// TIA Portal V20 export
TYPE "LBP_typeTMTurret"
TITLE = Tool management / Gestion des outils
// User data type for block LBP_TMTurret [DB73] / Type de données utilisateur pour bloc LBP_TMTurret [DB73]
   STRUCT
      IFNo : Array[1..16] of Bool;   // Interface [number] active / Interface [numéro] active
      Quit : Array[1..16] of Bool;   // Perform Quit-End / Effectuer Quit-End
      TIF : Array[1..16] of Struct
         Comp : Bool;   // Compulsory change / Modification obligatoire
         Perform : Bool;   // Perform change / Effectuer modification/changement
         f0_2 : Bool;   // Reserved / Réservé
         T0 : Bool;   // T0 programmed / T0 programmé
         f0_4 : Bool;   // Reserved / Réservé
         f0_5 : Bool;   // Reserved / Réservé
         ManTOut : Bool;   // Unload hand tool from spindle manually / Décharger manuellement l'outil manuel de la broche
         f0_7 : Bool;   // Reserved / Réservé
         PerfStatusError : Bool;   // Negative acknowledge / Acquittement négatif
         n1_1 : Bool;   // Reserved / Réservé
         n1_2 : Bool;   // Reserved / Réservé
         n1_3 : Bool;   // Reserved / Réservé
         n1_4 : Bool;   // Reserved / Réservé
         n1_5 : Bool;   // Reserved / Réservé
         n1_6 : Bool;   // Reserved / Réservé
         DataInDB1073 : Bool;   // Multitool data stored in DB1073 / Données Multitool enregistrées dans DB1073
         Channel : Byte;   // Assigned channel / Canal affecté
         TMNo : Byte;   // Tool management number / Numéro de gestion des outils
         VdiTcp0 : DInt;   // User parameter 0 / Variable utilisateur libre 0
         VdiTcp1 : DInt;   // User parameter 1 / Variable utilisateur libre 1
         VdiTcp2 : DInt;   // User parameter 2 / Variable utilisateur libre 2
         BufferIdent : Int;   // Reserved (buffer identification) / Réservé (identifiant tampon)
         BufferNo : Int;   // Rel. location in buffer (res.) / Emplacement relatif dans tampon (rés.)
         SMag : Int;   // Magazine number of turret / Numéro de magasin de la tourelle
         SLoc : Int;   // Location number for new tool / Numéro d'emplacement du nouvel outil
         TMag : Int;   // Magazine number of turret (res.) / Numéro de magasin de la tourelle (rés.)
         TLoc : Int;   // Location number for previous tool / Numéro d'emplacement de l'outil précédent
         LocType : Int;   // Tool new: location type / Nouvel outil : type d'emplacement
         SLeft : Int;   // Tool new: size left / Nouvel outil : taille côté gauche
         SRight : Int;   // Tool new: size right / Nouvel outil : taille côté droit
         STop : Int;   // Tool new: size top / Nouvel outil : taille dessus
         SBottom : Int;   // Tool new: size bottom / Nouvel outil : taille dessous
         TInBuffer : Bool;   // ID for tools in buffer / ID pour outils dans tampon
         IgnoreDisabled : Bool;   // Ignore disabled / Ignorer désactivation
         Unload : Bool;   // To be unloaded / À décharger
         Load : Bool;   // To be loaded / À charger
         MasterTool : Bool;   // Tool is the master tool / L'outil est un outil principal
         n38_5 : Bool;   // Reserved / Réservé
         Exchange_1to1 : Bool;   // 1:1 exchange / Échange 1:1
         HandTool : Bool;   // Hand tool / Outil manuel
         Active : Bool;   // Active tool / Outil actif
         Enabled : Bool;   // Tool enabled / Outil activé
         Disabled : Bool;   // Tool disabled / Outil désactivé
         Measured : Bool;   // Tool measured / Outil mesuré
         Prewarn : Bool;   // Prewarning limit reached / Seuil de préavis atteint
         Change : Bool;   // Tool being changed / Outil en cours de changement
         FixedLoc : Bool;   // Tool fixed location coded / Emplacement fixe d'outil codé
         Used : Bool;   // Tool was in use / Outil a été utilisé
         TNo : Int;   // Tool new: T number / Nouvel outil : numéro d'outil
         MyPlace : Int;   // Original location of new tool / Emplacement d'origine du nouvel outil
      END_STRUCT;
   END_STRUCT;
   // // TIF[2].Comp : Compulsory change / Modification obligatoire
   // // TIF[3].Comp : Compulsory change / Modification obligatoire
   // // TIF[4].Comp : Compulsory change / Modification obligatoire
   // // TIF[5].Comp : Compulsory change / Modification obligatoire
   // // TIF[6].Comp : Compulsory change / Modification obligatoire
   // // TIF[7].Comp : Compulsory change / Modification obligatoire
   // // TIF[8].Comp : Compulsory change / Modification obligatoire
   // // TIF[9].Comp : Compulsory change / Modification obligatoire
   // // TIF[10].Comp : Compulsory change / Modification obligatoire
   // // TIF[11].Comp : Compulsory change / Modification obligatoire
   // // TIF[12].Comp : Compulsory change / Modification obligatoire
   // // TIF[13].Comp : Compulsory change / Modification obligatoire
   // // TIF[14].Comp : Compulsory change / Modification obligatoire
   // // TIF[15].Comp : Compulsory change / Modification obligatoire
   // // TIF[16].Comp : Compulsory change / Modification obligatoire
   // // TIF[2].Perform : Perform change / Effectuer modification/changement
   // // TIF[3].Perform : Perform change / Effectuer modification/changement
   // // TIF[4].Perform : Perform change / Effectuer modification/changement
   // // TIF[5].Perform : Perform change / Effectuer modification/changement
   // // TIF[6].Perform : Perform change / Effectuer modification/changement
   // // TIF[7].Perform : Perform change / Effectuer modification/changement
   // // TIF[8].Perform : Perform change / Effectuer modification/changement
   // // TIF[9].Perform : Perform change / Effectuer modification/changement
   // // TIF[10].Perform : Perform change / Effectuer modification/changement
   // // TIF[11].Perform : Perform change / Effectuer modification/changement
   // // TIF[12].Perform : Perform change / Effectuer modification/changement
   // // TIF[13].Perform : Perform change / Effectuer modification/changement
   // // TIF[14].Perform : Perform change / Effectuer modification/changement
   // // TIF[15].Perform : Perform change / Effectuer modification/changement
   // // TIF[16].Perform : Perform change / Effectuer modification/changement
   // // TIF[2].f0_2 : Reserved / Réservé
   // // TIF[3].f0_2 : Reserved / Réservé
   // // TIF[4].f0_2 : Reserved / Réservé
   // // TIF[5].f0_2 : Reserved / Réservé
   // // TIF[6].f0_2 : Reserved / Réservé
   // // TIF[7].f0_2 : Reserved / Réservé
   // // TIF[8].f0_2 : Reserved / Réservé
   // // TIF[9].f0_2 : Reserved / Réservé
   // // TIF[10].f0_2 : Reserved / Réservé
   // // TIF[11].f0_2 : Reserved / Réservé
   // // TIF[12].f0_2 : Reserved / Réservé
   // // TIF[13].f0_2 : Reserved / Réservé
   // // TIF[14].f0_2 : Reserved / Réservé
   // // TIF[15].f0_2 : Reserved / Réservé
   // // TIF[16].f0_2 : Reserved / Réservé
   // // TIF[2].T0 : T0 programmed / T0 programmé
   // // TIF[3].T0 : T0 programmed / T0 programmé
   // // TIF[4].T0 : T0 programmed / T0 programmé
   // // TIF[5].T0 : T0 programmed / T0 programmé
   // // TIF[6].T0 : T0 programmed / T0 programmé
   // // TIF[7].T0 : T0 programmed / T0 programmé
   // // TIF[8].T0 : T0 programmed / T0 programmé
   // // TIF[9].T0 : T0 programmed / T0 programmé
   // // TIF[10].T0 : T0 programmed / T0 programmé
   // // TIF[11].T0 : T0 programmed / T0 programmé
   // // TIF[12].T0 : T0 programmed / T0 programmé
   // // TIF[13].T0 : T0 programmed / T0 programmé
   // // TIF[14].T0 : T0 programmed / T0 programmé
   // // TIF[15].T0 : T0 programmed / T0 programmé
   // // TIF[16].T0 : T0 programmed / T0 programmé
   // // TIF[2].f0_4 : Reserved / Réservé
   // // TIF[3].f0_4 : Reserved / Réservé
   // // TIF[4].f0_4 : Reserved / Réservé
   // // TIF[5].f0_4 : Reserved / Réservé
   // // TIF[6].f0_4 : Reserved / Réservé
   // // TIF[7].f0_4 : Reserved / Réservé
   // // TIF[8].f0_4 : Reserved / Réservé
   // // TIF[9].f0_4 : Reserved / Réservé
   // // TIF[10].f0_4 : Reserved / Réservé
   // // TIF[11].f0_4 : Reserved / Réservé
   // // TIF[12].f0_4 : Reserved / Réservé
   // // TIF[13].f0_4 : Reserved / Réservé
   // // TIF[14].f0_4 : Reserved / Réservé
   // // TIF[15].f0_4 : Reserved / Réservé
   // // TIF[16].f0_4 : Reserved / Réservé
   // // TIF[2].f0_5 : Reserved / Réservé
   // // TIF[3].f0_5 : Reserved / Réservé
   // // TIF[4].f0_5 : Reserved / Réservé
   // // TIF[5].f0_5 : Reserved / Réservé
   // // TIF[6].f0_5 : Reserved / Réservé
   // // TIF[7].f0_5 : Reserved / Réservé
   // // TIF[8].f0_5 : Reserved / Réservé
   // // TIF[9].f0_5 : Reserved / Réservé
   // // TIF[10].f0_5 : Reserved / Réservé
   // // TIF[11].f0_5 : Reserved / Réservé
   // // TIF[12].f0_5 : Reserved / Réservé
   // // TIF[13].f0_5 : Reserved / Réservé
   // // TIF[14].f0_5 : Reserved / Réservé
   // // TIF[15].f0_5 : Reserved / Réservé
   // // TIF[16].f0_5 : Reserved / Réservé
   // // TIF[2].ManTOut : Unload hand tool from spindle manually / Décharger manuellement l'outil manuel de la broche
   // // TIF[3].ManTOut : Unload hand tool from spindle manually / Décharger manuellement l'outil manuel de la broche
   // // TIF[4].ManTOut : Unload hand tool from spindle manually / Décharger manuellement l'outil manuel de la broche
   // // TIF[5].ManTOut : Unload hand tool from spindle manually / Décharger manuellement l'outil manuel de la broche
   // // TIF[6].ManTOut : Unload hand tool from spindle manually / Décharger manuellement l'outil manuel de la broche
   // // TIF[7].ManTOut : Unload hand tool from spindle manually / Décharger manuellement l'outil manuel de la broche
   // // TIF[8].ManTOut : Unload hand tool from spindle manually / Décharger manuellement l'outil manuel de la broche
   // // TIF[9].ManTOut : Unload hand tool from spindle manually / Décharger manuellement l'outil manuel de la broche
   // // TIF[10].ManTOut : Unload hand tool from spindle manually / Décharger manuellement l'outil manuel de la broche
   // // TIF[11].ManTOut : Unload hand tool from spindle manually / Décharger manuellement l'outil manuel de la broche
   // // TIF[12].ManTOut : Unload hand tool from spindle manually / Décharger manuellement l'outil manuel de la broche
   // // TIF[13].ManTOut : Unload hand tool from spindle manually / Décharger manuellement l'outil manuel de la broche
   // // TIF[14].ManTOut : Unload hand tool from spindle manually / Décharger manuellement l'outil manuel de la broche
   // // TIF[15].ManTOut : Unload hand tool from spindle manually / Décharger manuellement l'outil manuel de la broche
   // // TIF[16].ManTOut : Unload hand tool from spindle manually / Décharger manuellement l'outil manuel de la broche
   // // TIF[2].f0_7 : Reserved / Réservé
   // // TIF[3].f0_7 : Reserved / Réservé
   // // TIF[4].f0_7 : Reserved / Réservé
   // // TIF[5].f0_7 : Reserved / Réservé
   // // TIF[6].f0_7 : Reserved / Réservé
   // // TIF[7].f0_7 : Reserved / Réservé
   // // TIF[8].f0_7 : Reserved / Réservé
   // // TIF[9].f0_7 : Reserved / Réservé
   // // TIF[10].f0_7 : Reserved / Réservé
   // // TIF[11].f0_7 : Reserved / Réservé
   // // TIF[12].f0_7 : Reserved / Réservé
   // // TIF[13].f0_7 : Reserved / Réservé
   // // TIF[14].f0_7 : Reserved / Réservé
   // // TIF[15].f0_7 : Reserved / Réservé
   // // TIF[16].f0_7 : Reserved / Réservé
   // // TIF[2].PerfStatusError : Negative acknowledge / Acquittement négatif
   // // TIF[3].PerfStatusError : Negative acknowledge / Acquittement négatif
   // // TIF[4].PerfStatusError : Negative acknowledge / Acquittement négatif
   // // TIF[5].PerfStatusError : Negative acknowledge / Acquittement négatif
   // // TIF[6].PerfStatusError : Negative acknowledge / Acquittement négatif
   // // TIF[7].PerfStatusError : Negative acknowledge / Acquittement négatif
   // // TIF[8].PerfStatusError : Negative acknowledge / Acquittement négatif
   // // TIF[9].PerfStatusError : Negative acknowledge / Acquittement négatif
   // // TIF[10].PerfStatusError : Negative acknowledge / Acquittement négatif
   // // TIF[11].PerfStatusError : Negative acknowledge / Acquittement négatif
   // // TIF[12].PerfStatusError : Negative acknowledge / Acquittement négatif
   // // TIF[13].PerfStatusError : Negative acknowledge / Acquittement négatif
   // // TIF[14].PerfStatusError : Negative acknowledge / Acquittement négatif
   // // TIF[15].PerfStatusError : Negative acknowledge / Acquittement négatif
   // // TIF[16].PerfStatusError : Negative acknowledge / Acquittement négatif
   // // TIF[2].n1_1 : Reserved / Réservé
   // // TIF[3].n1_1 : Reserved / Réservé
   // // TIF[4].n1_1 : Reserved / Réservé
   // // TIF[5].n1_1 : Reserved / Réservé
   // // TIF[6].n1_1 : Reserved / Réservé
   // // TIF[7].n1_1 : Reserved / Réservé
   // // TIF[8].n1_1 : Reserved / Réservé
   // // TIF[9].n1_1 : Reserved / Réservé
   // // TIF[10].n1_1 : Reserved / Réservé
   // // TIF[11].n1_1 : Reserved / Réservé
   // // TIF[12].n1_1 : Reserved / Réservé
   // // TIF[13].n1_1 : Reserved / Réservé
   // // TIF[14].n1_1 : Reserved / Réservé
   // // TIF[15].n1_1 : Reserved / Réservé
   // // TIF[16].n1_1 : Reserved / Réservé
   // // TIF[2].n1_2 : Reserved / Réservé
   // // TIF[3].n1_2 : Reserved / Réservé
   // // TIF[4].n1_2 : Reserved / Réservé
   // // TIF[5].n1_2 : Reserved / Réservé
   // // TIF[6].n1_2 : Reserved / Réservé
   // // TIF[7].n1_2 : Reserved / Réservé
   // // TIF[8].n1_2 : Reserved / Réservé
   // // TIF[9].n1_2 : Reserved / Réservé
   // // TIF[10].n1_2 : Reserved / Réservé
   // // TIF[11].n1_2 : Reserved / Réservé
   // // TIF[12].n1_2 : Reserved / Réservé
   // // TIF[13].n1_2 : Reserved / Réservé
   // // TIF[14].n1_2 : Reserved / Réservé
   // // TIF[15].n1_2 : Reserved / Réservé
   // // TIF[16].n1_2 : Reserved / Réservé
   // // TIF[2].n1_3 : Reserved / Réservé
   // // TIF[3].n1_3 : Reserved / Réservé
   // // TIF[4].n1_3 : Reserved / Réservé
   // // TIF[5].n1_3 : Reserved / Réservé
   // // TIF[6].n1_3 : Reserved / Réservé
   // // TIF[7].n1_3 : Reserved / Réservé
   // // TIF[8].n1_3 : Reserved / Réservé
   // // TIF[9].n1_3 : Reserved / Réservé
   // // TIF[10].n1_3 : Reserved / Réservé
   // // TIF[11].n1_3 : Reserved / Réservé
   // // TIF[12].n1_3 : Reserved / Réservé
   // // TIF[13].n1_3 : Reserved / Réservé
   // // TIF[14].n1_3 : Reserved / Réservé
   // // TIF[15].n1_3 : Reserved / Réservé
   // // TIF[16].n1_3 : Reserved / Réservé
   // // TIF[2].n1_4 : Reserved / Réservé
   // // TIF[3].n1_4 : Reserved / Réservé
   // // TIF[4].n1_4 : Reserved / Réservé
   // // TIF[5].n1_4 : Reserved / Réservé
   // // TIF[6].n1_4 : Reserved / Réservé
   // // TIF[7].n1_4 : Reserved / Réservé
   // // TIF[8].n1_4 : Reserved / Réservé
   // // TIF[9].n1_4 : Reserved / Réservé
   // // TIF[10].n1_4 : Reserved / Réservé
   // // TIF[11].n1_4 : Reserved / Réservé
   // // TIF[12].n1_4 : Reserved / Réservé
   // // TIF[13].n1_4 : Reserved / Réservé
   // // TIF[14].n1_4 : Reserved / Réservé
   // // TIF[15].n1_4 : Reserved / Réservé
   // // TIF[16].n1_4 : Reserved / Réservé
   // // TIF[2].n1_5 : Reserved / Réservé
   // // TIF[3].n1_5 : Reserved / Réservé
   // // TIF[4].n1_5 : Reserved / Réservé
   // // TIF[5].n1_5 : Reserved / Réservé
   // // TIF[6].n1_5 : Reserved / Réservé
   // // TIF[7].n1_5 : Reserved / Réservé
   // // TIF[8].n1_5 : Reserved / Réservé
   // // TIF[9].n1_5 : Reserved / Réservé
   // // TIF[10].n1_5 : Reserved / Réservé
   // // TIF[11].n1_5 : Reserved / Réservé
   // // TIF[12].n1_5 : Reserved / Réservé
   // // TIF[13].n1_5 : Reserved / Réservé
   // // TIF[14].n1_5 : Reserved / Réservé
   // // TIF[15].n1_5 : Reserved / Réservé
   // // TIF[16].n1_5 : Reserved / Réservé
   // // TIF[2].n1_6 : Reserved / Réservé
   // // TIF[3].n1_6 : Reserved / Réservé
   // // TIF[4].n1_6 : Reserved / Réservé
   // // TIF[5].n1_6 : Reserved / Réservé
   // // TIF[6].n1_6 : Reserved / Réservé
   // // TIF[7].n1_6 : Reserved / Réservé
   // // TIF[8].n1_6 : Reserved / Réservé
   // // TIF[9].n1_6 : Reserved / Réservé
   // // TIF[10].n1_6 : Reserved / Réservé
   // // TIF[11].n1_6 : Reserved / Réservé
   // // TIF[12].n1_6 : Reserved / Réservé
   // // TIF[13].n1_6 : Reserved / Réservé
   // // TIF[14].n1_6 : Reserved / Réservé
   // // TIF[15].n1_6 : Reserved / Réservé
   // // TIF[16].n1_6 : Reserved / Réservé
   // // TIF[2].DataInDB1073 : Multitool data stored in DB1073 / Données Multitool enregistrées dans DB1073
   // // TIF[3].DataInDB1073 : Multitool data stored in DB1073 / Données Multitool enregistrées dans DB1073
   // // TIF[4].DataInDB1073 : Multitool data stored in DB1073 / Données Multitool enregistrées dans DB1073
   // // TIF[5].DataInDB1073 : Multitool data stored in DB1073 / Données Multitool enregistrées dans DB1073
   // // TIF[6].DataInDB1073 : Multitool data stored in DB1073 / Données Multitool enregistrées dans DB1073
   // // TIF[7].DataInDB1073 : Multitool data stored in DB1073 / Données Multitool enregistrées dans DB1073
   // // TIF[8].DataInDB1073 : Multitool data stored in DB1073 / Données Multitool enregistrées dans DB1073
   // // TIF[9].DataInDB1073 : Multitool data stored in DB1073 / Données Multitool enregistrées dans DB1073
   // // TIF[10].DataInDB1073 : Multitool data stored in DB1073 / Données Multitool enregistrées dans DB1073
   // // TIF[11].DataInDB1073 : Multitool data stored in DB1073 / Données Multitool enregistrées dans DB1073
   // // TIF[12].DataInDB1073 : Multitool data stored in DB1073 / Données Multitool enregistrées dans DB1073
   // // TIF[13].DataInDB1073 : Multitool data stored in DB1073 / Données Multitool enregistrées dans DB1073
   // // TIF[14].DataInDB1073 : Multitool data stored in DB1073 / Données Multitool enregistrées dans DB1073
   // // TIF[15].DataInDB1073 : Multitool data stored in DB1073 / Données Multitool enregistrées dans DB1073
   // // TIF[16].DataInDB1073 : Multitool data stored in DB1073 / Données Multitool enregistrées dans DB1073
   // // TIF[2].Channel : Assigned channel / Canal affecté
   // // TIF[3].Channel : Assigned channel / Canal affecté
   // // TIF[4].Channel : Assigned channel / Canal affecté
   // // TIF[5].Channel : Assigned channel / Canal affecté
   // // TIF[6].Channel : Assigned channel / Canal affecté
   // // TIF[7].Channel : Assigned channel / Canal affecté
   // // TIF[8].Channel : Assigned channel / Canal affecté
   // // TIF[9].Channel : Assigned channel / Canal affecté
   // // TIF[10].Channel : Assigned channel / Canal affecté
   // // TIF[11].Channel : Assigned channel / Canal affecté
   // // TIF[12].Channel : Assigned channel / Canal affecté
   // // TIF[13].Channel : Assigned channel / Canal affecté
   // // TIF[14].Channel : Assigned channel / Canal affecté
   // // TIF[15].Channel : Assigned channel / Canal affecté
   // // TIF[16].Channel : Assigned channel / Canal affecté
   // // TIF[2].TMNo : Tool management number / Numéro de gestion des outils
   // // TIF[3].TMNo : Tool management number / Numéro de gestion des outils
   // // TIF[4].TMNo : Tool management number / Numéro de gestion des outils
   // // TIF[5].TMNo : Tool management number / Numéro de gestion des outils
   // // TIF[6].TMNo : Tool management number / Numéro de gestion des outils
   // // TIF[7].TMNo : Tool management number / Numéro de gestion des outils
   // // TIF[8].TMNo : Tool management number / Numéro de gestion des outils
   // // TIF[9].TMNo : Tool management number / Numéro de gestion des outils
   // // TIF[10].TMNo : Tool management number / Numéro de gestion des outils
   // // TIF[11].TMNo : Tool management number / Numéro de gestion des outils
   // // TIF[12].TMNo : Tool management number / Numéro de gestion des outils
   // // TIF[13].TMNo : Tool management number / Numéro de gestion des outils
   // // TIF[14].TMNo : Tool management number / Numéro de gestion des outils
   // // TIF[15].TMNo : Tool management number / Numéro de gestion des outils
   // // TIF[16].TMNo : Tool management number / Numéro de gestion des outils
   // // TIF[2].VdiTcp0 : User parameter 0 / Variable utilisateur libre 0
   // // TIF[3].VdiTcp0 : User parameter 0 / Variable utilisateur libre 0
   // // TIF[4].VdiTcp0 : User parameter 0 / Variable utilisateur libre 0
   // // TIF[5].VdiTcp0 : User parameter 0 / Variable utilisateur libre 0
   // // TIF[6].VdiTcp0 : User parameter 0 / Variable utilisateur libre 0
   // // TIF[7].VdiTcp0 : User parameter 0 / Variable utilisateur libre 0
   // // TIF[8].VdiTcp0 : User parameter 0 / Variable utilisateur libre 0
   // // TIF[9].VdiTcp0 : User parameter 0 / Variable utilisateur libre 0
   // // TIF[10].VdiTcp0 : User parameter 0 / Variable utilisateur libre 0
   // // TIF[11].VdiTcp0 : User parameter 0 / Variable utilisateur libre 0
   // // TIF[12].VdiTcp0 : User parameter 0 / Variable utilisateur libre 0
   // // TIF[13].VdiTcp0 : User parameter 0 / Variable utilisateur libre 0
   // // TIF[14].VdiTcp0 : User parameter 0 / Variable utilisateur libre 0
   // // TIF[15].VdiTcp0 : User parameter 0 / Variable utilisateur libre 0
   // // TIF[16].VdiTcp0 : User parameter 0 / Variable utilisateur libre 0
   // // TIF[2].VdiTcp1 : User parameter 1 / Variable utilisateur libre 1
   // // TIF[3].VdiTcp1 : User parameter 1 / Variable utilisateur libre 1
   // // TIF[4].VdiTcp1 : User parameter 1 / Variable utilisateur libre 1
   // // TIF[5].VdiTcp1 : User parameter 1 / Variable utilisateur libre 1
   // // TIF[6].VdiTcp1 : User parameter 1 / Variable utilisateur libre 1
   // // TIF[7].VdiTcp1 : User parameter 1 / Variable utilisateur libre 1
   // // TIF[8].VdiTcp1 : User parameter 1 / Variable utilisateur libre 1
   // // TIF[9].VdiTcp1 : User parameter 1 / Variable utilisateur libre 1
   // // TIF[10].VdiTcp1 : User parameter 1 / Variable utilisateur libre 1
   // // TIF[11].VdiTcp1 : User parameter 1 / Variable utilisateur libre 1
   // // TIF[12].VdiTcp1 : User parameter 1 / Variable utilisateur libre 1
   // // TIF[13].VdiTcp1 : User parameter 1 / Variable utilisateur libre 1
   // // TIF[14].VdiTcp1 : User parameter 1 / Variable utilisateur libre 1
   // // TIF[15].VdiTcp1 : User parameter 1 / Variable utilisateur libre 1
   // // TIF[16].VdiTcp1 : User parameter 1 / Variable utilisateur libre 1
   // // TIF[2].VdiTcp2 : User parameter 2 / Variable utilisateur libre 2
   // // TIF[3].VdiTcp2 : User parameter 2 / Variable utilisateur libre 2
   // // TIF[4].VdiTcp2 : User parameter 2 / Variable utilisateur libre 2
   // // TIF[5].VdiTcp2 : User parameter 2 / Variable utilisateur libre 2
   // // TIF[6].VdiTcp2 : User parameter 2 / Variable utilisateur libre 2
   // // TIF[7].VdiTcp2 : User parameter 2 / Variable utilisateur libre 2
   // // TIF[8].VdiTcp2 : User parameter 2 / Variable utilisateur libre 2
   // // TIF[9].VdiTcp2 : User parameter 2 / Variable utilisateur libre 2
   // // TIF[10].VdiTcp2 : User parameter 2 / Variable utilisateur libre 2
   // // TIF[11].VdiTcp2 : User parameter 2 / Variable utilisateur libre 2
   // // TIF[12].VdiTcp2 : User parameter 2 / Variable utilisateur libre 2
   // // TIF[13].VdiTcp2 : User parameter 2 / Variable utilisateur libre 2
   // // TIF[14].VdiTcp2 : User parameter 2 / Variable utilisateur libre 2
   // // TIF[15].VdiTcp2 : User parameter 2 / Variable utilisateur libre 2
   // // TIF[16].VdiTcp2 : User parameter 2 / Variable utilisateur libre 2
   // // TIF[2].BufferIdent : Reserved (buffer identification) / Réservé (identifiant tampon)
   // // TIF[3].BufferIdent : Reserved (buffer identification) / Réservé (identifiant tampon)
   // // TIF[4].BufferIdent : Reserved (buffer identification) / Réservé (identifiant tampon)
   // // TIF[5].BufferIdent : Reserved (buffer identification) / Réservé (identifiant tampon)
   // // TIF[6].BufferIdent : Reserved (buffer identification) / Réservé (identifiant tampon)
   // // TIF[7].BufferIdent : Reserved (buffer identification) / Réservé (identifiant tampon)
   // // TIF[8].BufferIdent : Reserved (buffer identification) / Réservé (identifiant tampon)
   // // TIF[9].BufferIdent : Reserved (buffer identification) / Réservé (identifiant tampon)
   // // TIF[10].BufferIdent : Reserved (buffer identification) / Réservé (identifiant tampon)
   // // TIF[11].BufferIdent : Reserved (buffer identification) / Réservé (identifiant tampon)
   // // TIF[12].BufferIdent : Reserved (buffer identification) / Réservé (identifiant tampon)
   // // TIF[13].BufferIdent : Reserved (buffer identification) / Réservé (identifiant tampon)
   // // TIF[14].BufferIdent : Reserved (buffer identification) / Réservé (identifiant tampon)
   // // TIF[15].BufferIdent : Reserved (buffer identification) / Réservé (identifiant tampon)
   // // TIF[16].BufferIdent : Reserved (buffer identification) / Réservé (identifiant tampon)
   // // TIF[2].BufferNo : Rel. location in buffer (res.) / Emplacement relatif dans tampon (rés.)
   // // TIF[3].BufferNo : Rel. location in buffer (res.) / Emplacement relatif dans tampon (rés.)
   // // TIF[4].BufferNo : Rel. location in buffer (res.) / Emplacement relatif dans tampon (rés.)
   // // TIF[5].BufferNo : Rel. location in buffer (res.) / Emplacement relatif dans tampon (rés.)
   // // TIF[6].BufferNo : Rel. location in buffer (res.) / Emplacement relatif dans tampon (rés.)
   // // TIF[7].BufferNo : Rel. location in buffer (res.) / Emplacement relatif dans tampon (rés.)
   // // TIF[8].BufferNo : Rel. location in buffer (res.) / Emplacement relatif dans tampon (rés.)
   // // TIF[9].BufferNo : Rel. location in buffer (res.) / Emplacement relatif dans tampon (rés.)
   // // TIF[10].BufferNo : Rel. location in buffer (res.) / Emplacement relatif dans tampon (rés.)
   // // TIF[11].BufferNo : Rel. location in buffer (res.) / Emplacement relatif dans tampon (rés.)
   // // TIF[12].BufferNo : Rel. location in buffer (res.) / Emplacement relatif dans tampon (rés.)
   // // TIF[13].BufferNo : Rel. location in buffer (res.) / Emplacement relatif dans tampon (rés.)
   // // TIF[14].BufferNo : Rel. location in buffer (res.) / Emplacement relatif dans tampon (rés.)
   // // TIF[15].BufferNo : Rel. location in buffer (res.) / Emplacement relatif dans tampon (rés.)
   // // TIF[16].BufferNo : Rel. location in buffer (res.) / Emplacement relatif dans tampon (rés.)
   // // TIF[2].SMag : Magazine number of turret / Numéro de magasin de la tourelle
   // // TIF[3].SMag : Magazine number of turret / Numéro de magasin de la tourelle
   // // TIF[4].SMag : Magazine number of turret / Numéro de magasin de la tourelle
   // // TIF[5].SMag : Magazine number of turret / Numéro de magasin de la tourelle
   // // TIF[6].SMag : Magazine number of turret / Numéro de magasin de la tourelle
   // // TIF[7].SMag : Magazine number of turret / Numéro de magasin de la tourelle
   // // TIF[8].SMag : Magazine number of turret / Numéro de magasin de la tourelle
   // // TIF[9].SMag : Magazine number of turret / Numéro de magasin de la tourelle
   // // TIF[10].SMag : Magazine number of turret / Numéro de magasin de la tourelle
   // // TIF[11].SMag : Magazine number of turret / Numéro de magasin de la tourelle
   // // TIF[12].SMag : Magazine number of turret / Numéro de magasin de la tourelle
   // // TIF[13].SMag : Magazine number of turret / Numéro de magasin de la tourelle
   // // TIF[14].SMag : Magazine number of turret / Numéro de magasin de la tourelle
   // // TIF[15].SMag : Magazine number of turret / Numéro de magasin de la tourelle
   // // TIF[16].SMag : Magazine number of turret / Numéro de magasin de la tourelle
   // // TIF[2].SLoc : Location number for new tool / Numéro d'emplacement du nouvel outil
   // // TIF[3].SLoc : Location number for new tool / Numéro d'emplacement du nouvel outil
   // // TIF[4].SLoc : Location number for new tool / Numéro d'emplacement du nouvel outil
   // // TIF[5].SLoc : Location number for new tool / Numéro d'emplacement du nouvel outil
   // // TIF[6].SLoc : Location number for new tool / Numéro d'emplacement du nouvel outil
   // // TIF[7].SLoc : Location number for new tool / Numéro d'emplacement du nouvel outil
   // // TIF[8].SLoc : Location number for new tool / Numéro d'emplacement du nouvel outil
   // // TIF[9].SLoc : Location number for new tool / Numéro d'emplacement du nouvel outil
   // // TIF[10].SLoc : Location number for new tool / Numéro d'emplacement du nouvel outil
   // // TIF[11].SLoc : Location number for new tool / Numéro d'emplacement du nouvel outil
   // // TIF[12].SLoc : Location number for new tool / Numéro d'emplacement du nouvel outil
   // // TIF[13].SLoc : Location number for new tool / Numéro d'emplacement du nouvel outil
   // // TIF[14].SLoc : Location number for new tool / Numéro d'emplacement du nouvel outil
   // // TIF[15].SLoc : Location number for new tool / Numéro d'emplacement du nouvel outil
   // // TIF[16].SLoc : Location number for new tool / Numéro d'emplacement du nouvel outil
   // // TIF[2].TMag : Magazine number of turret (res.) / Numéro de magasin de la tourelle (rés.)
   // // TIF[3].TMag : Magazine number of turret (res.) / Numéro de magasin de la tourelle (rés.)
   // // TIF[4].TMag : Magazine number of turret (res.) / Numéro de magasin de la tourelle (rés.)
   // // TIF[5].TMag : Magazine number of turret (res.) / Numéro de magasin de la tourelle (rés.)
   // // TIF[6].TMag : Magazine number of turret (res.) / Numéro de magasin de la tourelle (rés.)
   // // TIF[7].TMag : Magazine number of turret (res.) / Numéro de magasin de la tourelle (rés.)
   // // TIF[8].TMag : Magazine number of turret (res.) / Numéro de magasin de la tourelle (rés.)
   // // TIF[9].TMag : Magazine number of turret (res.) / Numéro de magasin de la tourelle (rés.)
   // // TIF[10].TMag : Magazine number of turret (res.) / Numéro de magasin de la tourelle (rés.)
   // // TIF[11].TMag : Magazine number of turret (res.) / Numéro de magasin de la tourelle (rés.)
   // // TIF[12].TMag : Magazine number of turret (res.) / Numéro de magasin de la tourelle (rés.)
   // // TIF[13].TMag : Magazine number of turret (res.) / Numéro de magasin de la tourelle (rés.)
   // // TIF[14].TMag : Magazine number of turret (res.) / Numéro de magasin de la tourelle (rés.)
   // // TIF[15].TMag : Magazine number of turret (res.) / Numéro de magasin de la tourelle (rés.)
   // // TIF[16].TMag : Magazine number of turret (res.) / Numéro de magasin de la tourelle (rés.)
   // // TIF[2].TLoc : Location number for previous tool / Numéro d'emplacement de l'outil précédent
   // // TIF[3].TLoc : Location number for previous tool / Numéro d'emplacement de l'outil précédent
   // // TIF[4].TLoc : Location number for previous tool / Numéro d'emplacement de l'outil précédent
   // // TIF[5].TLoc : Location number for previous tool / Numéro d'emplacement de l'outil précédent
   // // TIF[6].TLoc : Location number for previous tool / Numéro d'emplacement de l'outil précédent
   // // TIF[7].TLoc : Location number for previous tool / Numéro d'emplacement de l'outil précédent
   // // TIF[8].TLoc : Location number for previous tool / Numéro d'emplacement de l'outil précédent
   // // TIF[9].TLoc : Location number for previous tool / Numéro d'emplacement de l'outil précédent
   // // TIF[10].TLoc : Location number for previous tool / Numéro d'emplacement de l'outil précédent
   // // TIF[11].TLoc : Location number for previous tool / Numéro d'emplacement de l'outil précédent
   // // TIF[12].TLoc : Location number for previous tool / Numéro d'emplacement de l'outil précédent
   // // TIF[13].TLoc : Location number for previous tool / Numéro d'emplacement de l'outil précédent
   // // TIF[14].TLoc : Location number for previous tool / Numéro d'emplacement de l'outil précédent
   // // TIF[15].TLoc : Location number for previous tool / Numéro d'emplacement de l'outil précédent
   // // TIF[16].TLoc : Location number for previous tool / Numéro d'emplacement de l'outil précédent
   // // TIF[2].LocType : Tool new: location type / Nouvel outil : type d'emplacement
   // // TIF[3].LocType : Tool new: location type / Nouvel outil : type d'emplacement
   // // TIF[4].LocType : Tool new: location type / Nouvel outil : type d'emplacement
   // // TIF[5].LocType : Tool new: location type / Nouvel outil : type d'emplacement
   // // TIF[6].LocType : Tool new: location type / Nouvel outil : type d'emplacement
   // // TIF[7].LocType : Tool new: location type / Nouvel outil : type d'emplacement
   // // TIF[8].LocType : Tool new: location type / Nouvel outil : type d'emplacement
   // // TIF[9].LocType : Tool new: location type / Nouvel outil : type d'emplacement
   // // TIF[10].LocType : Tool new: location type / Nouvel outil : type d'emplacement
   // // TIF[11].LocType : Tool new: location type / Nouvel outil : type d'emplacement
   // // TIF[12].LocType : Tool new: location type / Nouvel outil : type d'emplacement
   // // TIF[13].LocType : Tool new: location type / Nouvel outil : type d'emplacement
   // // TIF[14].LocType : Tool new: location type / Nouvel outil : type d'emplacement
   // // TIF[15].LocType : Tool new: location type / Nouvel outil : type d'emplacement
   // // TIF[16].LocType : Tool new: location type / Nouvel outil : type d'emplacement
   // // TIF[2].SLeft : Tool new: size left / Nouvel outil : taille côté gauche
   // // TIF[3].SLeft : Tool new: size left / Nouvel outil : taille côté gauche
   // // TIF[4].SLeft : Tool new: size left / Nouvel outil : taille côté gauche
   // // TIF[5].SLeft : Tool new: size left / Nouvel outil : taille côté gauche
   // // TIF[6].SLeft : Tool new: size left / Nouvel outil : taille côté gauche
   // // TIF[7].SLeft : Tool new: size left / Nouvel outil : taille côté gauche
   // // TIF[8].SLeft : Tool new: size left / Nouvel outil : taille côté gauche
   // // TIF[9].SLeft : Tool new: size left / Nouvel outil : taille côté gauche
   // // TIF[10].SLeft : Tool new: size left / Nouvel outil : taille côté gauche
   // // TIF[11].SLeft : Tool new: size left / Nouvel outil : taille côté gauche
   // // TIF[12].SLeft : Tool new: size left / Nouvel outil : taille côté gauche
   // // TIF[13].SLeft : Tool new: size left / Nouvel outil : taille côté gauche
   // // TIF[14].SLeft : Tool new: size left / Nouvel outil : taille côté gauche
   // // TIF[15].SLeft : Tool new: size left / Nouvel outil : taille côté gauche
   // // TIF[16].SLeft : Tool new: size left / Nouvel outil : taille côté gauche
   // // TIF[2].SRight : Tool new: size right / Nouvel outil : taille côté droit
   // // TIF[3].SRight : Tool new: size right / Nouvel outil : taille côté droit
   // // TIF[4].SRight : Tool new: size right / Nouvel outil : taille côté droit
   // // TIF[5].SRight : Tool new: size right / Nouvel outil : taille côté droit
   // // TIF[6].SRight : Tool new: size right / Nouvel outil : taille côté droit
   // // TIF[7].SRight : Tool new: size right / Nouvel outil : taille côté droit
   // // TIF[8].SRight : Tool new: size right / Nouvel outil : taille côté droit
   // // TIF[9].SRight : Tool new: size right / Nouvel outil : taille côté droit
   // // TIF[10].SRight : Tool new: size right / Nouvel outil : taille côté droit
   // // TIF[11].SRight : Tool new: size right / Nouvel outil : taille côté droit
   // // TIF[12].SRight : Tool new: size right / Nouvel outil : taille côté droit
   // // TIF[13].SRight : Tool new: size right / Nouvel outil : taille côté droit
   // // TIF[14].SRight : Tool new: size right / Nouvel outil : taille côté droit
   // // TIF[15].SRight : Tool new: size right / Nouvel outil : taille côté droit
   // // TIF[16].SRight : Tool new: size right / Nouvel outil : taille côté droit
   // // TIF[2].STop : Tool new: size top / Nouvel outil : taille dessus
   // // TIF[3].STop : Tool new: size top / Nouvel outil : taille dessus
   // // TIF[4].STop : Tool new: size top / Nouvel outil : taille dessus
   // // TIF[5].STop : Tool new: size top / Nouvel outil : taille dessus
   // // TIF[6].STop : Tool new: size top / Nouvel outil : taille dessus
   // // TIF[7].STop : Tool new: size top / Nouvel outil : taille dessus
   // // TIF[8].STop : Tool new: size top / Nouvel outil : taille dessus
   // // TIF[9].STop : Tool new: size top / Nouvel outil : taille dessus
   // // TIF[10].STop : Tool new: size top / Nouvel outil : taille dessus
   // // TIF[11].STop : Tool new: size top / Nouvel outil : taille dessus
   // // TIF[12].STop : Tool new: size top / Nouvel outil : taille dessus
   // // TIF[13].STop : Tool new: size top / Nouvel outil : taille dessus
   // // TIF[14].STop : Tool new: size top / Nouvel outil : taille dessus
   // // TIF[15].STop : Tool new: size top / Nouvel outil : taille dessus
   // // TIF[16].STop : Tool new: size top / Nouvel outil : taille dessus
   // // TIF[2].SBottom : Tool new: size bottom / Nouvel outil : taille dessous
   // // TIF[3].SBottom : Tool new: size bottom / Nouvel outil : taille dessous
   // // TIF[4].SBottom : Tool new: size bottom / Nouvel outil : taille dessous
   // // TIF[5].SBottom : Tool new: size bottom / Nouvel outil : taille dessous
   // // TIF[6].SBottom : Tool new: size bottom / Nouvel outil : taille dessous
   // // TIF[7].SBottom : Tool new: size bottom / Nouvel outil : taille dessous
   // // TIF[8].SBottom : Tool new: size bottom / Nouvel outil : taille dessous
   // // TIF[9].SBottom : Tool new: size bottom / Nouvel outil : taille dessous
   // // TIF[10].SBottom : Tool new: size bottom / Nouvel outil : taille dessous
   // // TIF[11].SBottom : Tool new: size bottom / Nouvel outil : taille dessous
   // // TIF[12].SBottom : Tool new: size bottom / Nouvel outil : taille dessous
   // // TIF[13].SBottom : Tool new: size bottom / Nouvel outil : taille dessous
   // // TIF[14].SBottom : Tool new: size bottom / Nouvel outil : taille dessous
   // // TIF[15].SBottom : Tool new: size bottom / Nouvel outil : taille dessous
   // // TIF[16].SBottom : Tool new: size bottom / Nouvel outil : taille dessous
   // // TIF[2].TInBuffer : ID for tools in buffer / ID pour outils dans tampon
   // // TIF[3].TInBuffer : ID for tools in buffer / ID pour outils dans tampon
   // // TIF[4].TInBuffer : ID for tools in buffer / ID pour outils dans tampon
   // // TIF[5].TInBuffer : ID for tools in buffer / ID pour outils dans tampon
   // // TIF[6].TInBuffer : ID for tools in buffer / ID pour outils dans tampon
   // // TIF[7].TInBuffer : ID for tools in buffer / ID pour outils dans tampon
   // // TIF[8].TInBuffer : ID for tools in buffer / ID pour outils dans tampon
   // // TIF[9].TInBuffer : ID for tools in buffer / ID pour outils dans tampon
   // // TIF[10].TInBuffer : ID for tools in buffer / ID pour outils dans tampon
   // // TIF[11].TInBuffer : ID for tools in buffer / ID pour outils dans tampon
   // // TIF[12].TInBuffer : ID for tools in buffer / ID pour outils dans tampon
   // // TIF[13].TInBuffer : ID for tools in buffer / ID pour outils dans tampon
   // // TIF[14].TInBuffer : ID for tools in buffer / ID pour outils dans tampon
   // // TIF[15].TInBuffer : ID for tools in buffer / ID pour outils dans tampon
   // // TIF[16].TInBuffer : ID for tools in buffer / ID pour outils dans tampon
   // // TIF[2].IgnoreDisabled : Ignore disabled / Ignorer désactivation
   // // TIF[3].IgnoreDisabled : Ignore disabled / Ignorer désactivation
   // // TIF[4].IgnoreDisabled : Ignore disabled / Ignorer désactivation
   // // TIF[5].IgnoreDisabled : Ignore disabled / Ignorer désactivation
   // // TIF[6].IgnoreDisabled : Ignore disabled / Ignorer désactivation
   // // TIF[7].IgnoreDisabled : Ignore disabled / Ignorer désactivation
   // // TIF[8].IgnoreDisabled : Ignore disabled / Ignorer désactivation
   // // TIF[9].IgnoreDisabled : Ignore disabled / Ignorer désactivation
   // // TIF[10].IgnoreDisabled : Ignore disabled / Ignorer désactivation
   // // TIF[11].IgnoreDisabled : Ignore disabled / Ignorer désactivation
   // // TIF[12].IgnoreDisabled : Ignore disabled / Ignorer désactivation
   // // TIF[13].IgnoreDisabled : Ignore disabled / Ignorer désactivation
   // // TIF[14].IgnoreDisabled : Ignore disabled / Ignorer désactivation
   // // TIF[15].IgnoreDisabled : Ignore disabled / Ignorer désactivation
   // // TIF[16].IgnoreDisabled : Ignore disabled / Ignorer désactivation
   // // TIF[2].Unload : To be unloaded / À décharger
   // // TIF[3].Unload : To be unloaded / À décharger
   // // TIF[4].Unload : To be unloaded / À décharger
   // // TIF[5].Unload : To be unloaded / À décharger
   // // TIF[6].Unload : To be unloaded / À décharger
   // // TIF[7].Unload : To be unloaded / À décharger
   // // TIF[8].Unload : To be unloaded / À décharger
   // // TIF[9].Unload : To be unloaded / À décharger
   // // TIF[10].Unload : To be unloaded / À décharger
   // // TIF[11].Unload : To be unloaded / À décharger
   // // TIF[12].Unload : To be unloaded / À décharger
   // // TIF[13].Unload : To be unloaded / À décharger
   // // TIF[14].Unload : To be unloaded / À décharger
   // // TIF[15].Unload : To be unloaded / À décharger
   // // TIF[16].Unload : To be unloaded / À décharger
   // // TIF[2].Load : To be loaded / À charger
   // // TIF[3].Load : To be loaded / À charger
   // // TIF[4].Load : To be loaded / À charger
   // // TIF[5].Load : To be loaded / À charger
   // // TIF[6].Load : To be loaded / À charger
   // // TIF[7].Load : To be loaded / À charger
   // // TIF[8].Load : To be loaded / À charger
   // // TIF[9].Load : To be loaded / À charger
   // // TIF[10].Load : To be loaded / À charger
   // // TIF[11].Load : To be loaded / À charger
   // // TIF[12].Load : To be loaded / À charger
   // // TIF[13].Load : To be loaded / À charger
   // // TIF[14].Load : To be loaded / À charger
   // // TIF[15].Load : To be loaded / À charger
   // // TIF[16].Load : To be loaded / À charger
   // // TIF[2].MasterTool : Tool is the master tool / L'outil est un outil principal
   // // TIF[3].MasterTool : Tool is the master tool / L'outil est un outil principal
   // // TIF[4].MasterTool : Tool is the master tool / L'outil est un outil principal
   // // TIF[5].MasterTool : Tool is the master tool / L'outil est un outil principal
   // // TIF[6].MasterTool : Tool is the master tool / L'outil est un outil principal
   // // TIF[7].MasterTool : Tool is the master tool / L'outil est un outil principal
   // // TIF[8].MasterTool : Tool is the master tool / L'outil est un outil principal
   // // TIF[9].MasterTool : Tool is the master tool / L'outil est un outil principal
   // // TIF[10].MasterTool : Tool is the master tool / L'outil est un outil principal
   // // TIF[11].MasterTool : Tool is the master tool / L'outil est un outil principal
   // // TIF[12].MasterTool : Tool is the master tool / L'outil est un outil principal
   // // TIF[13].MasterTool : Tool is the master tool / L'outil est un outil principal
   // // TIF[14].MasterTool : Tool is the master tool / L'outil est un outil principal
   // // TIF[15].MasterTool : Tool is the master tool / L'outil est un outil principal
   // // TIF[16].MasterTool : Tool is the master tool / L'outil est un outil principal
   // // TIF[2].n38_5 : Reserved / Réservé
   // // TIF[3].n38_5 : Reserved / Réservé
   // // TIF[4].n38_5 : Reserved / Réservé
   // // TIF[5].n38_5 : Reserved / Réservé
   // // TIF[6].n38_5 : Reserved / Réservé
   // // TIF[7].n38_5 : Reserved / Réservé
   // // TIF[8].n38_5 : Reserved / Réservé
   // // TIF[9].n38_5 : Reserved / Réservé
   // // TIF[10].n38_5 : Reserved / Réservé
   // // TIF[11].n38_5 : Reserved / Réservé
   // // TIF[12].n38_5 : Reserved / Réservé
   // // TIF[13].n38_5 : Reserved / Réservé
   // // TIF[14].n38_5 : Reserved / Réservé
   // // TIF[15].n38_5 : Reserved / Réservé
   // // TIF[16].n38_5 : Reserved / Réservé
   // // TIF[2].Exchange_1to1 : 1:1 exchange / Échange 1:1
   // // TIF[3].Exchange_1to1 : 1:1 exchange / Échange 1:1
   // // TIF[4].Exchange_1to1 : 1:1 exchange / Échange 1:1
   // // TIF[5].Exchange_1to1 : 1:1 exchange / Échange 1:1
   // // TIF[6].Exchange_1to1 : 1:1 exchange / Échange 1:1
   // // TIF[7].Exchange_1to1 : 1:1 exchange / Échange 1:1
   // // TIF[8].Exchange_1to1 : 1:1 exchange / Échange 1:1
   // // TIF[9].Exchange_1to1 : 1:1 exchange / Échange 1:1
   // // TIF[10].Exchange_1to1 : 1:1 exchange / Échange 1:1
   // // TIF[11].Exchange_1to1 : 1:1 exchange / Échange 1:1
   // // TIF[12].Exchange_1to1 : 1:1 exchange / Échange 1:1
   // // TIF[13].Exchange_1to1 : 1:1 exchange / Échange 1:1
   // // TIF[14].Exchange_1to1 : 1:1 exchange / Échange 1:1
   // // TIF[15].Exchange_1to1 : 1:1 exchange / Échange 1:1
   // // TIF[16].Exchange_1to1 : 1:1 exchange / Échange 1:1
   // // TIF[2].HandTool : Hand tool / Outil manuel
   // // TIF[3].HandTool : Hand tool / Outil manuel
   // // TIF[4].HandTool : Hand tool / Outil manuel
   // // TIF[5].HandTool : Hand tool / Outil manuel
   // // TIF[6].HandTool : Hand tool / Outil manuel
   // // TIF[7].HandTool : Hand tool / Outil manuel
   // // TIF[8].HandTool : Hand tool / Outil manuel
   // // TIF[9].HandTool : Hand tool / Outil manuel
   // // TIF[10].HandTool : Hand tool / Outil manuel
   // // TIF[11].HandTool : Hand tool / Outil manuel
   // // TIF[12].HandTool : Hand tool / Outil manuel
   // // TIF[13].HandTool : Hand tool / Outil manuel
   // // TIF[14].HandTool : Hand tool / Outil manuel
   // // TIF[15].HandTool : Hand tool / Outil manuel
   // // TIF[16].HandTool : Hand tool / Outil manuel
   // // TIF[2].Active : Active tool / Outil actif
   // // TIF[3].Active : Active tool / Outil actif
   // // TIF[4].Active : Active tool / Outil actif
   // // TIF[5].Active : Active tool / Outil actif
   // // TIF[6].Active : Active tool / Outil actif
   // // TIF[7].Active : Active tool / Outil actif
   // // TIF[8].Active : Active tool / Outil actif
   // // TIF[9].Active : Active tool / Outil actif
   // // TIF[10].Active : Active tool / Outil actif
   // // TIF[11].Active : Active tool / Outil actif
   // // TIF[12].Active : Active tool / Outil actif
   // // TIF[13].Active : Active tool / Outil actif
   // // TIF[14].Active : Active tool / Outil actif
   // // TIF[15].Active : Active tool / Outil actif
   // // TIF[16].Active : Active tool / Outil actif
   // // TIF[2].Enabled : Tool enabled / Outil activé
   // // TIF[3].Enabled : Tool enabled / Outil activé
   // // TIF[4].Enabled : Tool enabled / Outil activé
   // // TIF[5].Enabled : Tool enabled / Outil activé
   // // TIF[6].Enabled : Tool enabled / Outil activé
   // // TIF[7].Enabled : Tool enabled / Outil activé
   // // TIF[8].Enabled : Tool enabled / Outil activé
   // // TIF[9].Enabled : Tool enabled / Outil activé
   // // TIF[10].Enabled : Tool enabled / Outil activé
   // // TIF[11].Enabled : Tool enabled / Outil activé
   // // TIF[12].Enabled : Tool enabled / Outil activé
   // // TIF[13].Enabled : Tool enabled / Outil activé
   // // TIF[14].Enabled : Tool enabled / Outil activé
   // // TIF[15].Enabled : Tool enabled / Outil activé
   // // TIF[16].Enabled : Tool enabled / Outil activé
   // // TIF[2].Disabled : Tool disabled / Outil désactivé
   // // TIF[3].Disabled : Tool disabled / Outil désactivé
   // // TIF[4].Disabled : Tool disabled / Outil désactivé
   // // TIF[5].Disabled : Tool disabled / Outil désactivé
   // // TIF[6].Disabled : Tool disabled / Outil désactivé
   // // TIF[7].Disabled : Tool disabled / Outil désactivé
   // // TIF[8].Disabled : Tool disabled / Outil désactivé
   // // TIF[9].Disabled : Tool disabled / Outil désactivé
   // // TIF[10].Disabled : Tool disabled / Outil désactivé
   // // TIF[11].Disabled : Tool disabled / Outil désactivé
   // // TIF[12].Disabled : Tool disabled / Outil désactivé
   // // TIF[13].Disabled : Tool disabled / Outil désactivé
   // // TIF[14].Disabled : Tool disabled / Outil désactivé
   // // TIF[15].Disabled : Tool disabled / Outil désactivé
   // // TIF[16].Disabled : Tool disabled / Outil désactivé
   // // TIF[2].Measured : Tool measured / Outil mesuré
   // // TIF[3].Measured : Tool measured / Outil mesuré
   // // TIF[4].Measured : Tool measured / Outil mesuré
   // // TIF[5].Measured : Tool measured / Outil mesuré
   // // TIF[6].Measured : Tool measured / Outil mesuré
   // // TIF[7].Measured : Tool measured / Outil mesuré
   // // TIF[8].Measured : Tool measured / Outil mesuré
   // // TIF[9].Measured : Tool measured / Outil mesuré
   // // TIF[10].Measured : Tool measured / Outil mesuré
   // // TIF[11].Measured : Tool measured / Outil mesuré
   // // TIF[12].Measured : Tool measured / Outil mesuré
   // // TIF[13].Measured : Tool measured / Outil mesuré
   // // TIF[14].Measured : Tool measured / Outil mesuré
   // // TIF[15].Measured : Tool measured / Outil mesuré
   // // TIF[16].Measured : Tool measured / Outil mesuré
   // // TIF[2].Prewarn : Prewarning limit reached / Seuil de préavis atteint
   // // TIF[3].Prewarn : Prewarning limit reached / Seuil de préavis atteint
   // // TIF[4].Prewarn : Prewarning limit reached / Seuil de préavis atteint
   // // TIF[5].Prewarn : Prewarning limit reached / Seuil de préavis atteint
   // // TIF[6].Prewarn : Prewarning limit reached / Seuil de préavis atteint
   // // TIF[7].Prewarn : Prewarning limit reached / Seuil de préavis atteint
   // // TIF[8].Prewarn : Prewarning limit reached / Seuil de préavis atteint
   // // TIF[9].Prewarn : Prewarning limit reached / Seuil de préavis atteint
   // // TIF[10].Prewarn : Prewarning limit reached / Seuil de préavis atteint
   // // TIF[11].Prewarn : Prewarning limit reached / Seuil de préavis atteint
   // // TIF[12].Prewarn : Prewarning limit reached / Seuil de préavis atteint
   // // TIF[13].Prewarn : Prewarning limit reached / Seuil de préavis atteint
   // // TIF[14].Prewarn : Prewarning limit reached / Seuil de préavis atteint
   // // TIF[15].Prewarn : Prewarning limit reached / Seuil de préavis atteint
   // // TIF[16].Prewarn : Prewarning limit reached / Seuil de préavis atteint
   // // TIF[2].Change : Tool being changed / Outil en cours de changement
   // // TIF[3].Change : Tool being changed / Outil en cours de changement
   // // TIF[4].Change : Tool being changed / Outil en cours de changement
   // // TIF[5].Change : Tool being changed / Outil en cours de changement
   // // TIF[6].Change : Tool being changed / Outil en cours de changement
   // // TIF[7].Change : Tool being changed / Outil en cours de changement
   // // TIF[8].Change : Tool being changed / Outil en cours de changement
   // // TIF[9].Change : Tool being changed / Outil en cours de changement
   // // TIF[10].Change : Tool being changed / Outil en cours de changement
   // // TIF[11].Change : Tool being changed / Outil en cours de changement
   // // TIF[12].Change : Tool being changed / Outil en cours de changement
   // // TIF[13].Change : Tool being changed / Outil en cours de changement
   // // TIF[14].Change : Tool being changed / Outil en cours de changement
   // // TIF[15].Change : Tool being changed / Outil en cours de changement
   // // TIF[16].Change : Tool being changed / Outil en cours de changement
   // // TIF[2].FixedLoc : Tool fixed location coded / Emplacement fixe d'outil codé
   // // TIF[3].FixedLoc : Tool fixed location coded / Emplacement fixe d'outil codé
   // // TIF[4].FixedLoc : Tool fixed location coded / Emplacement fixe d'outil codé
   // // TIF[5].FixedLoc : Tool fixed location coded / Emplacement fixe d'outil codé
   // // TIF[6].FixedLoc : Tool fixed location coded / Emplacement fixe d'outil codé
   // // TIF[7].FixedLoc : Tool fixed location coded / Emplacement fixe d'outil codé
   // // TIF[8].FixedLoc : Tool fixed location coded / Emplacement fixe d'outil codé
   // // TIF[9].FixedLoc : Tool fixed location coded / Emplacement fixe d'outil codé
   // // TIF[10].FixedLoc : Tool fixed location coded / Emplacement fixe d'outil codé
   // // TIF[11].FixedLoc : Tool fixed location coded / Emplacement fixe d'outil codé
   // // TIF[12].FixedLoc : Tool fixed location coded / Emplacement fixe d'outil codé
   // // TIF[13].FixedLoc : Tool fixed location coded / Emplacement fixe d'outil codé
   // // TIF[14].FixedLoc : Tool fixed location coded / Emplacement fixe d'outil codé
   // // TIF[15].FixedLoc : Tool fixed location coded / Emplacement fixe d'outil codé
   // // TIF[16].FixedLoc : Tool fixed location coded / Emplacement fixe d'outil codé
   // // TIF[2].Used : Tool was in use / Outil a été utilisé
   // // TIF[3].Used : Tool was in use / Outil a été utilisé
   // // TIF[4].Used : Tool was in use / Outil a été utilisé
   // // TIF[5].Used : Tool was in use / Outil a été utilisé
   // // TIF[6].Used : Tool was in use / Outil a été utilisé
   // // TIF[7].Used : Tool was in use / Outil a été utilisé
   // // TIF[8].Used : Tool was in use / Outil a été utilisé
   // // TIF[9].Used : Tool was in use / Outil a été utilisé
   // // TIF[10].Used : Tool was in use / Outil a été utilisé
   // // TIF[11].Used : Tool was in use / Outil a été utilisé
   // // TIF[12].Used : Tool was in use / Outil a été utilisé
   // // TIF[13].Used : Tool was in use / Outil a été utilisé
   // // TIF[14].Used : Tool was in use / Outil a été utilisé
   // // TIF[15].Used : Tool was in use / Outil a été utilisé
   // // TIF[16].Used : Tool was in use / Outil a été utilisé
   // // TIF[2].TNo : Tool new: T number / Nouvel outil : numéro d'outil
   // // TIF[3].TNo : Tool new: T number / Nouvel outil : numéro d'outil
   // // TIF[4].TNo : Tool new: T number / Nouvel outil : numéro d'outil
   // // TIF[5].TNo : Tool new: T number / Nouvel outil : numéro d'outil
   // // TIF[6].TNo : Tool new: T number / Nouvel outil : numéro d'outil
   // // TIF[7].TNo : Tool new: T number / Nouvel outil : numéro d'outil
   // // TIF[8].TNo : Tool new: T number / Nouvel outil : numéro d'outil
   // // TIF[9].TNo : Tool new: T number / Nouvel outil : numéro d'outil
   // // TIF[10].TNo : Tool new: T number / Nouvel outil : numéro d'outil
   // // TIF[11].TNo : Tool new: T number / Nouvel outil : numéro d'outil
   // // TIF[12].TNo : Tool new: T number / Nouvel outil : numéro d'outil
   // // TIF[13].TNo : Tool new: T number / Nouvel outil : numéro d'outil
   // // TIF[14].TNo : Tool new: T number / Nouvel outil : numéro d'outil
   // // TIF[15].TNo : Tool new: T number / Nouvel outil : numéro d'outil
   // // TIF[16].TNo : Tool new: T number / Nouvel outil : numéro d'outil
   // // TIF[2].MyPlace : Original location of new tool / Emplacement d'origine du nouvel outil
   // // TIF[3].MyPlace : Original location of new tool / Emplacement d'origine du nouvel outil
   // // TIF[4].MyPlace : Original location of new tool / Emplacement d'origine du nouvel outil
   // // TIF[5].MyPlace : Original location of new tool / Emplacement d'origine du nouvel outil
   // // TIF[6].MyPlace : Original location of new tool / Emplacement d'origine du nouvel outil
   // // TIF[7].MyPlace : Original location of new tool / Emplacement d'origine du nouvel outil
   // // TIF[8].MyPlace : Original location of new tool / Emplacement d'origine du nouvel outil
   // // TIF[9].MyPlace : Original location of new tool / Emplacement d'origine du nouvel outil
   // // TIF[10].MyPlace : Original location of new tool / Emplacement d'origine du nouvel outil
   // // TIF[11].MyPlace : Original location of new tool / Emplacement d'origine du nouvel outil
   // // TIF[12].MyPlace : Original location of new tool / Emplacement d'origine du nouvel outil
   // // TIF[13].MyPlace : Original location of new tool / Emplacement d'origine du nouvel outil
   // // TIF[14].MyPlace : Original location of new tool / Emplacement d'origine du nouvel outil
   // // TIF[15].MyPlace : Original location of new tool / Emplacement d'origine du nouvel outil
   // // TIF[16].MyPlace : Original location of new tool / Emplacement d'origine du nouvel outil
END_TYPE
